TYPE MOD_InputBelt_Q_stMotor :
STRUCT
	Command : INT;
	MoveLeft : BOOL;
	MoveRight : BOOL;
END_STRUCT
END_TYPE

(* stored: Version 1.1.0.1, ProductVersion 3.1.4024.6
   DUT MOD_InputBelt_Q_stMotor: Id {a627231d-3f0c-4ba3-8401-c74d85b13290} *)
